VAR_GLOBAL
		stDutData_Cnc1					: ST_Dut_Data;
END_VAR

(* stored: Version 1.1.0.1, ProductVersion 3.1.4024.12
   GVL GVL_CNC1: Id {8fde1a5d-a85b-45e8-991d-5a4aaeac6303} *)
